{attribute 'qualified_only'}
{attribute 'strict'}
{attribute 'to_string'}
TYPE E_PROCESS_CTRL :
(
  PROCESS_INIT              := 10,
  PROCESS_DISABLE           := 20,
  PROCESS_ENABLE            := 30,
  PROCESS_STATIONS_INFEED,

  PROCESS_STATIONS_ENTER    := 40,
  PROCESS_STATIONS_SEND,

  PROCESS_START             := 60,
  PROCESS_DONE              := 70,
  PROCESS_STATIONS_OUTFEED  := 80
);
END_TYPE

(* stored: Version 1.1.0.1, ProductVersion 3.1.4026.12
   DUT E_PROCESS_CTRL: Id {104b6d53-82e0-43bb-822e-312fbaf3fe62} *)
